SPLINE
SPL {X  -158.898, Y  +690.164, Z    +0.000, E1   +18.236, E3 -481675.354}
SPL {X  -159.149, Y  +687.882, Z    +0.000, E1   +16.368, E3 -481682.641}
SPL {X  -159.987, Y  +672.488, Z    +0.000, E1    +5.638, E3 -481704.183}
SPL {X  -159.990, Y  +663.928, Z    +0.000, E1    -0.338, E3 -481709.978}
SPL {X  -159.990, Y  +658.009, Z    +0.000, E1    -4.774, E3 -481713.678}
SPL {X  -159.990, Y  +651.567, Z    +0.000, E1    -9.674, E3 -481719.081}
SPL {X  -159.990, Y  +637.762, Z    +0.000, E1   -18.345, E3 -481736.439}
SPL {X  -159.990, Y  +626.382, Z    +0.000, E1   -22.040, E3 -481768.488}
SPL {X  -159.990, Y  +623.760, Z    +0.000, E1   -22.031, E3 -481782.266}
SPL {X  -159.990, Y  +621.334, Z    +0.000, E1   -22.029, E3 -481794.993}
SPL {X  -159.990, Y  +619.505, Z    +0.000, E1   -22.018, E3 -481804.608}
SPL {X  -159.990, Y  +617.621, Z    +0.000, E1   -22.025, E3 -481814.474}
SPL {X  -159.990, Y  +615.830, Z    +0.000, E1   -22.023, E3 -481823.874}
SPL {X  -159.990, Y  +614.007, Z    +0.000, E1   -22.018, E3 -481833.452}
SPL {X  -159.990, Y  +611.459, Z    +0.000, E1   -22.053, E3 -481846.738}
SPL {X  -159.990, Y  +608.810, Z    +0.000, E1   -22.023, E3 -481860.706}
SPL {X  -159.990, Y  +606.481, Z    +0.000, E1   -22.033, E3 -481872.882}
SPL {X  -159.990, Y  +603.419, Z    +0.000, E1   -22.064, E3 -481888.821}
SPL {X  -159.990, Y  +600.642, Z    +0.000, E1   -22.032, E3 -481903.451}
SPL {X  -159.990, Y  +598.568, Z    +0.000, E1   -22.046, E3 -481914.243}
SPL {X  -159.990, Y  +596.440, Z    +0.000, E1   -22.036, E3 -481925.425}
SPL {X  -159.990, Y  +593.768, Z    +0.000, E1   -22.071, E3 -481939.358}
SPL {X  -159.990, Y  +590.068, Z    +0.000, E1   -22.076, E3 -481958.726}
SPL {X  -159.990, Y  +587.130, Z    +0.000, E1   -22.046, E3 -481974.163}
SPL {X  -159.990, Y  +585.120, Z    +0.000, E1   -22.045, E3 -481984.665}
SPL {X  -159.990, Y  +583.118, Z    +0.000, E1   -22.052, E3 -481995.151}
SPL {X  -159.990, Y  +580.862, Z    +0.000, E1   -22.049, E3 -482006.989}
SPL {X  -159.990, Y  +578.386, Z    +0.000, E1   -22.057, E3 -482019.944}
SPL {X  -159.990, Y  +576.252, Z    +0.000, E1   -22.038, E3 -482031.168}
SPL {X  -159.990, Y  +574.280, Z    +0.000, E1   -22.051, E3 -482041.462}
SPL {X  -159.990, Y  +571.711, Z    +0.000, E1   -22.058, E3 -482054.935}
SPL {X  -159.990, Y  +569.285, Z    +0.000, E1   -22.044, E3 -482067.660}
SPL {X  -159.990, Y  +567.211, Z    +0.000, E1   -22.046, E3 -482078.522}
SPL {X  -159.990, Y  +565.039, Z    +0.000, E1   -22.047, E3 -482089.899}
SPL {X  -159.990, Y  +562.755, Z    +0.000, E1   -22.047, E3 -482101.884}
SPL {X  -159.990, Y  +559.661, Z    +0.000, E1   -22.078, E3 -482118.016}
SPL {X  -159.990, Y  +555.965, Z    +0.000, E1   -22.085, E3 -482137.325}
SPL {X  -159.990, Y  +553.115, Z    +0.000, E1   -22.054, E3 -482152.311}
SPL {X  -159.990, Y  +550.886, Z    +0.000, E1   -22.056, E3 -482163.992}
SPL {X  -159.990, Y  +547.986, Z    +0.000, E1   -22.078, E3 -482179.111}
SPL {X  -159.990, Y  +545.350, Z    +0.000, E1   -22.053, E3 -482192.973}
SPL {X  -159.990, Y  +543.405, Z    +0.000, E1   -22.048, E3 -482203.186}
SPL {X  -159.990, Y  +541.673, Z    +0.000, E1   -22.053, E3 -482212.249}
SPL {X  -159.990, Y  +539.341, Z    +0.000, E1   -22.056, E3 -482224.455}
SPL {X  -159.990, Y  +536.301, Z    +0.000, E1   -22.084, E3 -482240.309}
SPL {X  -159.990, Y  +533.389, Z    +0.000, E1   -22.057, E3 -482255.617}
SPL {X  -159.990, Y  +531.347, Z    +0.000, E1   -22.052, E3 -482266.317}
SPL {X  -159.990, Y  +529.626, Z    +0.000, E1   -22.051, E3 -482275.315}
SPL {X  -159.990, Y  +527.412, Z    +0.000, E1   -22.067, E3 -482286.867}
SPL {X  -159.990, Y  +524.425, Z    +0.000, E1   -22.078, E3 -482302.500}
SPL {X  -159.990, Y  +521.599, Z    +0.000, E1   -22.060, E3 -482317.342}
SPL {X  -159.990, Y  +519.209, Z    +0.000, E1   -22.063, E3 -482329.817}
SPL {X  -159.990, Y  +516.651, Z    +0.000, E1   -22.071, E3 -482343.196}
SPL {X  -159.990, Y  +514.122, Z    +0.000, E1   -22.061, E3 -482356.468}
SPL {X  -159.990, Y  +511.670, Z    +0.000, E1   -22.064, E3 -482369.318}
SPL {X  -159.990, Y  +506.947, Z    +0.000, E1   -23.726, E3 -482379.347}
SPL {X  -159.990, Y  +496.921, Z    +0.000, E1   -28.340, E3 -482388.095}
SPL {X  -159.990, Y  +495.822, Z    +0.000, E1   -27.449, E3 -482398.843}
SPL {X  -159.990, Y  +494.952, Z    +0.000, E1   -26.628, E3 -482408.426}
SPL {X  -159.990, Y  +493.896, Z    +0.000, E1   -25.736, E3 -482419.756}
SPL {X  -159.990, Y  +491.647, Z    +0.000, E1   -25.401, E3 -482432.291}
SPL {X  -159.990, Y  +488.807, Z    +0.000, E1   -25.397, E3 -482444.990}
SPL {X  -159.990, Y  +486.070, Z    +0.000, E1   -25.399, E3 -482457.221}
SPL {X  -159.990, Y  +483.747, Z    +0.000, E1   -25.384, E3 -482467.634}
SPL {X  -159.990, Y  +481.038, Z    +0.000, E1   -25.412, E3 -482479.689}
SPL {X  -159.990, Y  +478.407, Z    +0.000, E1   -25.384, E3 -482491.503}
SPL {X  -159.990, Y  +475.940, Z    +0.000, E1   -25.403, E3 -482502.493}
SPL {X  -159.990, Y  +473.026, Z    +0.000, E1   -25.399, E3 -482515.523}
SPL {X  -159.990, Y  +470.047, Z    +0.000, E1   -25.402, E3 -482528.842}
SPL {X  -159.990, Y  +467.082, Z    +0.000, E1   -25.399, E3 -482542.089}
SPL {X  -159.990, Y  +464.919, Z    +0.000, E1   -25.381, E3 -482551.815}
SPL {X  -159.990, Y  +462.520, Z    +0.000, E1   -25.400, E3 -482562.490}
SPL {X  -159.990, Y  +460.081, Z    +0.000, E1   -25.390, E3 -482573.391}
SPL {X  -159.990, Y  +457.497, Z    +0.000, E1   -25.403, E3 -482584.916}
SPL {X  -159.990, Y  +454.323, Z    +0.000, E1   -25.412, E3 -482599.075}
SPL {X  -159.990, Y  +450.823, Z    +0.000, E1   -25.417, E3 -482614.704}
SPL {X  -159.990, Y  +446.894, Z    +0.000, E1   -25.428, E3 -482632.261}
SPL {X  -159.990, Y  +443.345, Z    +0.000, E1   -25.390, E3 -482648.268}
SPL {X  -159.990, Y  +441.077, Z    +0.000, E1   -25.369, E3 -482658.466}
SPL {X  -159.990, Y  +438.608, Z    +0.000, E1   -25.392, E3 -482669.463}
SPL {X  -159.990, Y  +435.579, Z    +0.000, E1   -25.386, E3 -482683.017}
SPL {X  -159.990, Y  +432.613, Z    +0.000, E1   -25.390, E3 -482696.285}
SPL {X  -159.990, Y  +429.079, Z    +0.000, E1   -25.407, E3 -482712.055}
SPL {X  -159.990, Y  +426.149, Z    +0.000, E1   -25.374, E3 -482725.217}
SPL {X  -159.990, Y  +423.417, Z    +0.000, E1   -25.400, E3 -482737.383}
SPL {X  -159.990, Y  +420.283, Z    +0.000, E1   -25.386, E3 -482751.427}
SPL {X  -159.990, Y  +417.514, Z    +0.000, E1   -25.386, E3 -482763.812}
SPL {X  -159.990, Y  +414.805, Z    +0.000, E1   -25.385, E3 -482775.932}
SPL {X  -159.990, Y  +411.282, Z    +0.000, E1   -25.413, E3 -482791.632}
SPL {X  -159.990, Y  +407.450, Z    +0.000, E1   -25.401, E3 -482808.782}
SPL {X  -159.990, Y  +403.513, Z    +0.000, E1   -25.420, E3 -482826.335}
SPL {X  -159.990, Y  +399.257, Z    +0.000, E1   -25.420, E3 -482845.376}
SPL {X  -159.990, Y  +395.992, Z    +0.000, E1   -25.380, E3 -482860.066}
SPL {X  -159.990, Y  +393.569, Z    +0.000, E1   -25.379, E3 -482870.909}
SPL {X  -159.990, Y  +390.564, Z    +0.000, E1   -25.393, E3 -482884.353}
SPL {X  -159.990, Y  +387.503, Z    +0.000, E1   -25.378, E3 -482898.068}
SPL {X  -159.990, Y  +384.900, Z    +0.000, E1   -25.383, E3 -482909.678}
SPL {X  -159.990, Y  +382.110, Z    +0.000, E1   -25.393, E3 -482922.124}
SPL {X  -159.961, Y  +379.439, Z    +0.000, E1   -25.380, E3 -482934.103}
SPL {X  -159.894, Y  +376.959, Z    +0.000, E1   -25.370, E3 -482945.281}
SPL {X  -159.784, Y  +374.382, Z    +0.000, E1   -25.356, E3 -482956.921}
SPL {X  -159.621, Y  +371.640, Z    +0.000, E1   -25.335, E3 -482969.361}
SPL {X  -159.406, Y  +368.844, Z    +0.000, E1   -25.307, E3 -482982.074}
SPL {X  -159.144, Y  +366.072, Z    +0.000, E1   -25.281, E3 -482994.682}
SPL {X  -158.822, Y  +363.200, Z    +0.000, E1   -25.236, E3 -483007.855}
SPL {X  -158.491, Y  +360.654, Z    +0.000, E1   -25.188, E3 -483019.595}
SPL {X  -158.127, Y  +358.155, Z    +0.000, E1   -25.126, E3 -483031.214}
SPL {X  -158.095, Y  +357.947, Z    +0.000, E1   -21.741, E3 -483062.786}
ENDSPLINE

SPLINE
SPL {X  -158.454, Y  +360.384, Z    +0.000, E1   -19.366, E3 -483074.937}
SPL {X  -159.737, Y  +373.507, Z    +0.000, E1   -10.311, E3 -483096.973}
SPL {X  -159.990, Y  +382.574, Z    +0.000, E1    -4.463, E3 -483103.661}
SPL {X  -159.990, Y  +387.496, Z    +0.000, E1    -1.004, E3 -483106.406}
SPL {X  -159.990, Y  +395.121, Z    +0.000, E1    +4.514, E3 -483110.718}
SPL {X  -159.990, Y  +407.941, Z    +0.000, E1   +14.126, E3 -483122.792}
SPL {X  -159.990, Y  +418.671, Z    +0.000, E1   +19.855, E3 -483142.208}
SPL {X  -159.990, Y  +429.878, Z    +0.000, E1   +23.330, E3 -483172.264}
SPL {X  -159.990, Y  +432.103, Z    +0.000, E1   +23.301, E3 -483183.282}
SPL {X  -159.990, Y  +434.188, Z    +0.000, E1   +23.325, E3 -483193.479}
SPL {X  -159.990, Y  +436.320, Z    +0.000, E1   +23.304, E3 -483204.031}
SPL {X  -159.990, Y  +439.169, Z    +0.000, E1   +23.353, E3 -483217.948}
SPL {X  -159.990, Y  +442.945, Z    +0.000, E1   +23.339, E3 -483236.566}
SPL {X  -159.990, Y  +446.037, Z    +0.000, E1   +23.324, E3 -483251.816}
SPL {X  -159.990, Y  +448.797, Z    +0.000, E1   +23.331, E3 -483265.347}
SPL {X  -159.990, Y  +451.747, Z    +0.000, E1   +23.333, E3 -483279.895}
SPL {X  -159.990, Y  +455.185, Z    +0.000, E1   +23.350, E3 -483296.755}
SPL {X  -159.990, Y  +458.265, Z    +0.000, E1   +23.328, E3 -483311.941}
SPL {X  -159.990, Y  +460.492, Z    +0.000, E1   +23.317, E3 -483322.940}
SPL {X  -159.990, Y  +462.929, Z    +0.000, E1   +23.331, E3 -483334.896}
SPL {X  -159.990, Y  +465.027, Z    +0.000, E1   +23.313, E3 -483345.249}
SPL {X  -159.990, Y  +466.881, Z    +0.000, E1   +23.322, E3 -483354.359}
SPL {X  -159.990, Y  +468.951, Z    +0.000, E1   +23.319, E3 -483364.551}
SPL {X  -159.990, Y  +471.818, Z    +0.000, E1   +23.351, E3 -483378.597}
SPL {X  -159.990, Y  +474.801, Z    +0.000, E1   +23.320, E3 -483393.373}
SPL {X  -159.990, Y  +476.830, Z    +0.000, E1   +23.323, E3 -483403.352}
SPL {X  -159.990, Y  +479.553, Z    +0.000, E1   +23.328, E3 -483416.754}
SPL {X  -159.990, Y  +481.893, Z    +0.000, E1   +23.312, E3 -483428.304}
SPL {X  -159.990, Y  +483.782, Z    +0.000, E1   +23.316, E3 -483437.590}
SPL {X  -159.990, Y  +486.109, Z    +0.000, E1   +23.322, E3 -483449.042}
SPL {X  -159.990, Y  +489.247, Z    +0.000, E1   +23.348, E3 -483464.430}
SPL {X  -159.990, Y  +493.031, Z    +0.000, E1   +23.350, E3 -483483.054}
SPL {X  -159.990, Y  +496.869, Z    +0.000, E1   +23.349, E3 -483501.944}
SPL {X  -159.990, Y  +499.995, Z    +0.000, E1   +23.324, E3 -483517.377}
SPL {X  -159.990, Y  +502.456, Z    +0.000, E1   +23.324, E3 -483529.492}
SPL {X  -159.990, Y  +505.646, Z    +0.000, E1   +23.350, E3 -483545.147}
SPL {X  -159.990, Y  +508.862, Z    +0.000, E1   +23.328, E3 -483561.011}
SPL {X  -159.990, Y  +510.971, Z    +0.000, E1   +23.308, E3 -483571.439}
SPL {X  -159.990, Y  +512.484, Z    +0.000, E1   +23.309, E3 -483578.888}
SPL {X  -159.990, Y  +514.757, Z    +0.000, E1   +23.329, E3 -483590.041}
SPL {X  -159.990, Y  +517.536, Z    +0.000, E1   +23.326, E3 -483603.707}
SPL {X  -159.990, Y  +519.961, Z    +0.000, E1   +23.334, E3 -483615.560}
SPL {X  -159.990, Y  +521.849, Z    +0.000, E1   +23.320, E3 -483624.882}
SPL {X  -159.990, Y  +523.968, Z    +0.000, E1   +23.332, E3 -483635.318}
SPL {X  -159.990, Y  +526.466, Z    +0.000, E1   +23.320, E3 -483647.662}
SPL {X  -159.990, Y  +528.815, Z    +0.000, E1   +23.322, E3 -483659.221}
SPL {X  -159.990, Y  +531.246, Z    +0.000, E1   +23.325, E3 -483671.160}
SPL {X  -159.990, Y  +533.354, Z    +0.000, E1   +23.318, E3 -483681.545}
SPL {X  -159.990, Y  +534.931, Z    +0.000, E1   +23.312, E3 -483689.339}
SPL {X  -159.990, Y  +537.024, Z    +0.000, E1   +23.321, E3 -483699.638}
SPL {X  -159.990, Y  +539.129, Z    +0.000, E1   +23.310, E3 -483710.021}
SPL {X  -159.990, Y  +541.183, Z    +0.000, E1   +23.319, E3 -483720.118}
SPL {X  -159.990, Y  +544.314, Z    +0.000, E1   +23.352, E3 -483735.446}
SPL {X  -159.990, Y  +548.126, Z    +0.000, E1   +23.354, E3 -483754.201}
SPL {X  -159.990, Y  +551.344, Z    +0.000, E1   +23.327, E3 -483770.093}
SPL {X  -159.990, Y  +553.642, Z    +0.000, E1   +23.319, E3 -483781.412}
SPL {X  -159.990, Y  +556.481, Z    +0.000, E1   +23.354, E3 -483795.319}
SPL {X  -159.990, Y  +559.475, Z    +0.000, E1   +23.321, E3 -483810.125}
SPL {X  -159.990, Y  +561.830, Z    +0.000, E1   +23.325, E3 -483821.709}
SPL {X  -159.990, Y  +564.273, Z    +0.000, E1   +23.325, E3 -483833.733}
SPL {X  -159.990, Y  +566.342, Z    +0.000, E1   +23.314, E3 -483843.938}
SPL {X  -159.990, Y  +568.849, Z    +0.000, E1   +23.338, E3 -483856.233}
SPL {X  -159.990, Y  +572.204, Z    +0.000, E1   +23.344, E3 -483872.728}
SPL {X  -159.990, Y  +575.097, Z    +0.000, E1   +23.325, E3 -483887.005}
SPL {X  -159.990, Y  +577.540, Z    +0.000, E1   +23.325, E3 -483899.034}
SPL {X  -159.990, Y  +580.312, Z    +0.000, E1   +23.340, E3 -483912.615}
SPL {X  -159.990, Y  +583.018, Z    +0.000, E1   +23.331, E3 -483925.920}
SPL {X  -159.990, Y  +585.165, Z    +0.000, E1   +23.322, E3 -483936.536}
SPL {X  -159.990, Y  +587.388, Z    +0.000, E1   +23.328, E3 -483947.448}
SPL {X  -159.990, Y  +589.763, Z    +0.000, E1   +23.328, E3 -483959.135}
SPL {X  -159.990, Y  +592.397, Z    +0.000, E1   +23.344, E3 -483972.016}
SPL {X  -159.990, Y  +594.928, Z    +0.000, E1   +23.334, E3 -483984.478}
SPL {X  -159.990, Y  +597.981, Z    +0.000, E1   +23.373, E3 -483999.393}
SPL {X  -159.990, Y  +600.935, Z    +0.000, E1   +23.343, E3 -484013.926}
SPL {X  -159.990, Y  +603.047, Z    +0.000, E1   +23.344, E3 -484024.311}
SPL {X  -159.990, Y  +605.187, Z    +0.000, E1   +23.344, E3 -484034.833}
SPL {X  -159.990, Y  +607.319, Z    +0.000, E1   +23.353, E3 -484045.295}
SPL {X  -159.990, Y  +610.569, Z    +0.000, E1   +23.372, E3 -484061.260}
SPL {X  -159.990, Y  +613.591, Z    +0.000, E1   +23.342, E3 -484076.189}
SPL {X  -159.990, Y  +615.604, Z    +0.000, E1   +23.330, E3 -484086.127}
SPL {X  -159.990, Y  +618.445, Z    +0.000, E1   +23.368, E3 -484100.040}
SPL {X  -159.990, Y  +621.517, Z    +0.000, E1   +23.337, E3 -484115.204}
SPL {X  -159.990, Y  +623.764, Z    +0.000, E1   +23.335, E3 -484126.255}
SPL {X  -159.990, Y  +625.941, Z    +0.000, E1   +23.337, E3 -484136.946}
SPL {X  -159.990, Y  +628.611, Z    +0.000, E1   +23.357, E3 -484150.025}
SPL {X  -159.990, Y  +631.169, Z    +0.000, E1   +23.338, E3 -484162.629}
SPL {X  -159.990, Y  +633.318, Z    +0.000, E1   +23.339, E3 -484173.218}
SPL {X  -159.990, Y  +635.650, Z    +0.000, E1   +23.339, E3 -484184.689}
SPL {X  -159.990, Y  +637.839, Z    +0.000, E1   +23.335, E3 -484195.500}
SPL {X  -159.990, Y  +640.072, Z    +0.000, E1   +23.325, E3 -484206.532}
SPL {X  -159.990, Y  +642.230, Z    +0.000, E1   +23.323, E3 -484217.213}
SPL {X  -159.990, Y  +645.287, Z    +0.000, E1   +23.340, E3 -484232.239}
SPL {X  -159.990, Y  +648.792, Z    +0.000, E1   +23.346, E3 -484249.498}
SPL {X  -159.990, Y  +652.623, Z    +0.000, E1   +23.348, E3 -484268.333}
SPL {X  -159.990, Y  +656.380, Z    +0.000, E1   +23.347, E3 -484286.827}
SPL {X  -159.990, Y  +659.180, Z    +0.000, E1   +23.314, E3 -484300.676}
SPL {X  -159.990, Y  +661.392, Z    +0.000, E1   +23.318, E3 -484311.569}
SPL {X  -159.990, Y  +663.662, Z    +0.000, E1   +23.322, E3 -484322.693}
SPL {X  -159.990, Y  +665.964, Z    +0.000, E1   +23.328, E3 -484333.984}
SPL {X  -159.990, Y  +668.989, Z    +0.000, E1   +23.359, E3 -484348.820}
SPL {X  -159.983, Y  +672.946, Z    +0.000, E1   +23.359, E3 -484368.301}
SPL {X  -159.924, Y  +676.110, Z    +0.000, E1   +23.320, E3 -484384.000}
SPL {X  -159.845, Y  +678.302, Z    +0.000, E1   +23.298, E3 -484394.902}
SPL {X  -159.760, Y  +680.081, Z    +0.000, E1   +23.288, E3 -484403.746}
SPL {X  -159.626, Y  +682.287, Z    +0.000, E1   +23.280, E3 -484414.717}
SPL {X  -159.462, Y  +684.486, Z    +0.000, E1   +23.258, E3 -484425.717}
SPL {X  -159.246, Y  +686.911, Z    +0.000, E1   +23.230, E3 -484437.878}
SPL {X  -159.019, Y  +689.098, Z    +0.000, E1   +23.200, E3 -484448.880}
SPL {X  -158.771, Y  +691.210, Z    +0.000, E1   +23.159, E3 -484459.555}
SPL {X  -158.553, Y  +692.896, Z    +0.000, E1   +23.130, E3 -484468.085}
ENDSPLINE

SPLINE
SPL {X  -158.898, Y  +690.164, Z    +0.000, E1   +18.236, E3 -484501.441}
SPL {X  -159.149, Y  +687.882, Z    +0.000, E1   +16.368, E3 -484508.728}
SPL {X  -159.987, Y  +672.488, Z    +0.000, E1    +5.638, E3 -484530.270}
SPL {X  -159.990, Y  +663.928, Z    +0.000, E1    -0.338, E3 -484536.065}
SPL {X  -159.990, Y  +658.009, Z    +0.000, E1    -4.774, E3 -484539.765}
SPL {X  -159.990, Y  +651.567, Z    +0.000, E1    -9.674, E3 -484545.168}
SPL {X  -159.990, Y  +638.711, Z    +0.000, E1   -17.883, E3 -484560.814}
SPL {X  -159.990, Y  +631.642, Z    +0.000, E1   -20.884, E3 -484576.373}
SPL {X  -159.990, Y  +626.048, Z    +0.000, E1   -22.026, E3 -484596.366}
SPL {X  -159.990, Y  +623.760, Z    +0.000, E1   -22.031, E3 -484608.353}
SPL {X  -159.990, Y  +621.334, Z    +0.000, E1   -22.029, E3 -484621.080}
SPL {X  -159.990, Y  +619.505, Z    +0.000, E1   -22.018, E3 -484630.695}
SPL {X  -159.990, Y  +617.621, Z    +0.000, E1   -22.025, E3 -484640.561}
SPL {X  -159.990, Y  +615.830, Z    +0.000, E1   -22.023, E3 -484649.961}
SPL {X  -159.990, Y  +613.034, Z    +0.000, E1   -22.053, E3 -484664.568}
SPL {X  -159.990, Y  +609.503, Z    +0.000, E1   -22.054, E3 -484683.094}
SPL {X  -159.990, Y  +605.804, Z    +0.000, E1   -22.064, E3 -484702.438}
SPL {X  -159.990, Y  +602.819, Z    +0.000, E1   -22.037, E3 -484718.110}
SPL {X  -159.990, Y  +600.642, Z    +0.000, E1   -22.032, E3 -484729.538}
SPL {X  -159.990, Y  +598.568, Z    +0.000, E1   -22.046, E3 -484740.330}
SPL {X  -159.990, Y  +595.493, Z    +0.000, E1   -22.070, E3 -484756.414}
SPL {X  -159.990, Y  +592.865, Z    +0.000, E1   -22.036, E3 -484770.242}
SPL {X  -159.990, Y  +590.803, Z    +0.000, E1   -22.046, E3 -484781.033}
SPL {X  -159.990, Y  +587.778, Z    +0.000, E1   -22.073, E3 -484796.808}
SPL {X  -159.990, Y  +585.120, Z    +0.000, E1   -22.045, E3 -484810.752}
SPL {X  -159.990, Y  +583.118, Z    +0.000, E1   -22.052, E3 -484821.238}
SPL {X  -159.990, Y  +580.131, Z    +0.000, E1   -22.078, E3 -484836.845}
SPL {X  -159.990, Y  +576.888, Z    +0.000, E1   -22.061, E3 -484853.875}
SPL {X  -159.990, Y  +574.280, Z    +0.000, E1   -22.051, E3 -484867.549}
SPL {X  -159.990, Y  +572.375, Z    +0.000, E1   -22.037, E3 -484877.587}
SPL {X  -159.990, Y  +569.881, Z    +0.000, E1   -22.067, E3 -484890.581}
SPL {X  -159.990, Y  +567.211, Z    +0.000, E1   -22.046, E3 -484904.609}
SPL {X  -159.990, Y  +565.039, Z    +0.000, E1   -22.047, E3 -484915.986}
SPL {X  -159.990, Y  +562.755, Z    +0.000, E1   -22.047, E3 -484927.971}
SPL {X  -159.990, Y  +559.661, Z    +0.000, E1   -22.078, E3 -484944.103}
SPL {X  -159.990, Y  +555.965, Z    +0.000, E1   -22.085, E3 -484963.412}
SPL {X  -159.990, Y  +553.115, Z    +0.000, E1   -22.054, E3 -484978.398}
SPL {X  -159.990, Y  +550.886, Z    +0.000, E1   -22.056, E3 -484990.079}
SPL {X  -159.990, Y  +547.986, Z    +0.000, E1   -22.078, E3 -485005.198}
SPL {X  -159.990, Y  +545.350, Z    +0.000, E1   -22.053, E3 -485019.060}
SPL {X  -159.990, Y  +543.405, Z    +0.000, E1   -22.048, E3 -485029.273}
SPL {X  -159.990, Y  +541.673, Z    +0.000, E1   -22.053, E3 -485038.336}
SPL {X  -159.990, Y  +539.341, Z    +0.000, E1   -22.056, E3 -485050.542}
SPL {X  -159.990, Y  +536.301, Z    +0.000, E1   -22.084, E3 -485066.396}
SPL {X  -159.990, Y  +533.389, Z    +0.000, E1   -22.057, E3 -485081.704}
SPL {X  -159.990, Y  +530.476, Z    +0.000, E1   -22.084, E3 -485096.891}
SPL {X  -159.990, Y  +527.412, Z    +0.000, E1   -22.067, E3 -485112.954}
SPL {X  -159.990, Y  +525.349, Z    +0.000, E1   -22.050, E3 -485123.795}
SPL {X  -159.990, Y  +523.717, Z    +0.000, E1   -22.050, E3 -485132.361}
SPL {X  -159.990, Y  +521.599, Z    +0.000, E1   -22.060, E3 -485143.429}
SPL {X  -159.990, Y  +519.209, Z    +0.000, E1   -22.063, E3 -485155.904}
SPL {X  -159.990, Y  +517.330, Z    +0.000, E1   -22.053, E3 -485165.760}
SPL {X  -159.990, Y  +514.729, Z    +0.000, E1   -22.089, E3 -485179.318}
SPL {X  -159.990, Y  +511.670, Z    +0.000, E1   -22.064, E3 -485195.405}
SPL {X  -159.990, Y  +506.947, Z    +0.000, E1   -23.726, E3 -485205.434}
SPL {X  -159.990, Y  +496.921, Z    +0.000, E1   -28.340, E3 -485214.182}
SPL {X  -159.990, Y  +495.822, Z    +0.000, E1   -27.449, E3 -485224.930}
SPL {X  -159.990, Y  +494.952, Z    +0.000, E1   -26.628, E3 -485234.513}
SPL {X  -159.990, Y  +493.896, Z    +0.000, E1   -25.736, E3 -485245.843}
SPL {X  -159.990, Y  +491.647, Z    +0.000, E1   -25.401, E3 -485258.378}
SPL {X  -159.990, Y  +488.807, Z    +0.000, E1   -25.397, E3 -485271.077}
SPL {X  -159.990, Y  +486.070, Z    +0.000, E1   -25.399, E3 -485283.308}
SPL {X  -159.990, Y  +482.821, Z    +0.000, E1   -25.411, E3 -485297.809}
SPL {X  -159.990, Y  +480.183, Z    +0.000, E1   -25.384, E3 -485309.650}
SPL {X  -159.990, Y  +477.508, Z    +0.000, E1   -25.410, E3 -485321.558}
SPL {X  -159.990, Y  +473.634, Z    +0.000, E1   -25.426, E3 -485338.848}
SPL {X  -159.990, Y  +470.047, Z    +0.000, E1   -25.402, E3 -485354.928}
SPL {X  -159.990, Y  +466.213, Z    +0.000, E1   -25.433, E3 -485372.008}
SPL {X  -159.990, Y  +462.520, Z    +0.000, E1   -25.400, E3 -485388.577}
SPL {X  -159.990, Y  +460.081, Z    +0.000, E1   -25.390, E3 -485399.478}
SPL {X  -159.990, Y  +457.497, Z    +0.000, E1   -25.403, E3 -485411.003}
SPL {X  -159.990, Y  +455.126, Z    +0.000, E1   -25.389, E3 -485421.611}
SPL {X  -159.990, Y  +452.123, Z    +0.000, E1   -25.426, E3 -485434.969}
SPL {X  -159.990, Y  +448.503, Z    +0.000, E1   -25.410, E3 -485451.170}
SPL {X  -159.990, Y  +445.882, Z    +0.000, E1   -25.385, E3 -485462.973}
SPL {X  -159.990, Y  +443.345, Z    +0.000, E1   -25.390, E3 -485474.355}
SPL {X  -159.990, Y  +441.077, Z    +0.000, E1   -25.369, E3 -485484.553}
SPL {X  -159.990, Y  +438.608, Z    +0.000, E1   -25.392, E3 -485495.550}
SPL {X  -159.990, Y  +434.852, Z    +0.000, E1   -25.415, E3 -485512.305}
SPL {X  -159.990, Y  +430.645, Z    +0.000, E1   -25.414, E3 -485531.124}
SPL {X  -159.990, Y  +426.865, Z    +0.000, E1   -25.398, E3 -485548.054}
SPL {X  -159.990, Y  +424.251, Z    +0.000, E1   -25.375, E3 -485559.791}
SPL {X  -159.990, Y  +421.010, Z    +0.000, E1   -25.418, E3 -485574.206}
SPL {X  -159.990, Y  +417.514, Z    +0.000, E1   -25.386, E3 -485589.899}
SPL {X  -159.990, Y  +414.805, Z    +0.000, E1   -25.385, E3 -485602.019}
SPL {X  -159.990, Y  +411.282, Z    +0.000, E1   -25.413, E3 -485617.719}
SPL {X  -159.990, Y  +408.351, Z    +0.000, E1   -25.372, E3 -485630.906}
SPL {X  -159.990, Y  +405.773, Z    +0.000, E1   -25.398, E3 -485642.359}
SPL {X  -159.990, Y  +402.805, Z    +0.000, E1   -25.389, E3 -485655.645}
SPL {X  -159.990, Y  +400.083, Z    +0.000, E1   -25.388, E3 -485667.822}
SPL {X  -159.990, Y  +396.740, Z    +0.000, E1   -25.410, E3 -485682.746}
SPL {X  -159.990, Y  +392.622, Z    +0.000, E1   -25.413, E3 -485701.174}
SPL {X  -159.990, Y  +388.328, Z    +0.000, E1   -25.413, E3 -485720.402}
SPL {X  -159.990, Y  +384.900, Z    +0.000, E1   -25.383, E3 -485735.764}
SPL {X  -159.990, Y  +382.110, Z    +0.000, E1   -25.393, E3 -485748.211}
SPL {X  -159.961, Y  +379.439, Z    +0.000, E1   -25.380, E3 -485760.190}
SPL {X  -159.894, Y  +376.959, Z    +0.000, E1   -25.370, E3 -485771.368}
SPL {X  -159.784, Y  +374.382, Z    +0.000, E1   -25.356, E3 -485783.008}
SPL {X  -159.621, Y  +371.640, Z    +0.000, E1   -25.335, E3 -485795.448}
SPL {X  -159.406, Y  +368.844, Z    +0.000, E1   -25.307, E3 -485808.161}
SPL {X  -159.144, Y  +366.072, Z    +0.000, E1   -25.281, E3 -485820.769}
SPL {X  -158.822, Y  +363.200, Z    +0.000, E1   -25.236, E3 -485833.941}
SPL {X  -158.491, Y  +360.654, Z    +0.000, E1   -25.188, E3 -485845.682}
SPL {X  -158.127, Y  +358.155, Z    +0.000, E1   -25.126, E3 -485857.301}
SPL {X  -158.095, Y  +357.947, Z    +0.000, E1   -21.741, E3 -485888.873}
ENDSPLINE

SPLINE
SPL {X  -158.454, Y  +360.384, Z    +0.000, E1   -19.366, E3 -485901.024}
SPL {X  -159.737, Y  +373.507, Z    +0.000, E1   -10.311, E3 -485923.060}
SPL {X  -159.990, Y  +382.574, Z    +0.000, E1    -4.463, E3 -485929.748}
SPL {X  -159.990, Y  +389.909, Z    +0.000, E1    +0.662, E3 -485933.762}
SPL {X  -159.990, Y  +396.289, Z    +0.000, E1    +5.500, E3 -485937.542}
SPL {X  -159.990, Y  +407.941, Z    +0.000, E1   +14.126, E3 -485948.879}
SPL {X  -159.990, Y  +418.671, Z    +0.000, E1   +19.855, E3 -485968.295}
SPL {X  -159.990, Y  +429.878, Z    +0.000, E1   +23.330, E3 -485998.350}
SPL {X  -159.990, Y  +432.103, Z    +0.000, E1   +23.301, E3 -486009.369}
SPL {X  -159.990, Y  +434.188, Z    +0.000, E1   +23.325, E3 -486019.566}
SPL {X  -159.990, Y  +437.007, Z    +0.000, E1   +23.323, E3 -486033.457}
SPL {X  -159.990, Y  +439.778, Z    +0.000, E1   +23.323, E3 -486047.089}
SPL {X  -159.990, Y  +442.010, Z    +0.000, E1   +23.308, E3 -486058.110}
SPL {X  -159.990, Y  +443.729, Z    +0.000, E1   +23.310, E3 -486066.566}
SPL {X  -159.990, Y  +446.037, Z    +0.000, E1   +23.324, E3 -486077.903}
SPL {X  -159.990, Y  +449.434, Z    +0.000, E1   +23.356, E3 -486094.525}
SPL {X  -159.990, Y  +453.256, Z    +0.000, E1   +23.349, E3 -486113.360}
SPL {X  -159.990, Y  +455.953, Z    +0.000, E1   +23.320, E3 -486126.674}
SPL {X  -159.990, Y  +458.265, Z    +0.000, E1   +23.328, E3 -486138.028}
SPL {X  -159.990, Y  +461.258, Z    +0.000, E1   +23.344, E3 -486152.744}
SPL {X  -159.990, Y  +464.382, Z    +0.000, E1   +23.332, E3 -486168.126}
SPL {X  -159.990, Y  +466.881, Z    +0.000, E1   +23.322, E3 -486180.446}
SPL {X  -159.990, Y  +468.951, Z    +0.000, E1   +23.319, E3 -486190.638}
SPL {X  -159.990, Y  +470.991, Z    +0.000, E1   +23.322, E3 -486200.668}
SPL {X  -159.990, Y  +474.027, Z    +0.000, E1   +23.352, E3 -486215.571}
SPL {X  -159.990, Y  +477.600, Z    +0.000, E1   +23.351, E3 -486233.175}
SPL {X  -159.990, Y  +481.169, Z    +0.000, E1   +23.337, E3 -486250.772}
SPL {X  -159.990, Y  +483.782, Z    +0.000, E1   +23.316, E3 -486263.677}
SPL {X  -159.990, Y  +486.109, Z    +0.000, E1   +23.322, E3 -486275.129}
SPL {X  -159.990, Y  +489.247, Z    +0.000, E1   +23.348, E3 -486290.517}
SPL {X  -159.990, Y  +493.031, Z    +0.000, E1   +23.350, E3 -486309.141}
SPL {X  -159.990, Y  +496.869, Z    +0.000, E1   +23.349, E3 -486328.031}
SPL {X  -159.990, Y  +499.995, Z    +0.000, E1   +23.324, E3 -486343.464}
SPL {X  -159.990, Y  +502.456, Z    +0.000, E1   +23.324, E3 -486355.579}
SPL {X  -159.990, Y  +505.646, Z    +0.000, E1   +23.350, E3 -486371.234}
SPL {X  -159.990, Y  +508.862, Z    +0.000, E1   +23.328, E3 -486387.098}
SPL {X  -159.990, Y  +510.971, Z    +0.000, E1   +23.308, E3 -486397.526}
SPL {X  -159.990, Y  +513.289, Z    +0.000, E1   +23.332, E3 -486408.893}
SPL {X  -159.990, Y  +516.860, Z    +0.000, E1   +23.355, E3 -486426.410}
SPL {X  -159.990, Y  +520.719, Z    +0.000, E1   +23.363, E3 -486445.320}
SPL {X  -159.990, Y  +523.968, Z    +0.000, E1   +23.332, E3 -486461.405}
SPL {X  -159.990, Y  +526.466, Z    +0.000, E1   +23.320, E3 -486473.748}
SPL {X  -159.990, Y  +528.815, Z    +0.000, E1   +23.322, E3 -486485.308}
SPL {X  -159.990, Y  +531.246, Z    +0.000, E1   +23.325, E3 -486497.247}
SPL {X  -159.990, Y  +534.143, Z    +0.000, E1   +23.341, E3 -486511.482}
SPL {X  -159.990, Y  +537.024, Z    +0.000, E1   +23.321, E3 -486525.725}
SPL {X  -159.990, Y  +539.129, Z    +0.000, E1   +23.310, E3 -486536.108}
SPL {X  -159.990, Y  +541.882, Z    +0.000, E1   +23.346, E3 -486549.589}
SPL {X  -159.990, Y  +544.941, Z    +0.000, E1   +23.325, E3 -486564.671}
SPL {X  -159.990, Y  +547.390, Z    +0.000, E1   +23.325, E3 -486576.725}
SPL {X  -159.990, Y  +550.708, Z    +0.000, E1   +23.357, E3 -486592.992}
SPL {X  -159.990, Y  +553.642, Z    +0.000, E1   +23.319, E3 -486607.499}
SPL {X  -159.990, Y  +555.637, Z    +0.000, E1   +23.323, E3 -486617.313}
SPL {X  -159.990, Y  +558.758, Z    +0.000, E1   +23.351, E3 -486632.623}
SPL {X  -159.990, Y  +561.830, Z    +0.000, E1   +23.325, E3 -486647.796}
SPL {X  -159.990, Y  +564.273, Z    +0.000, E1   +23.325, E3 -486659.820}
SPL {X  -159.990, Y  +567.351, Z    +0.000, E1   +23.348, E3 -486674.916}
SPL {X  -159.990, Y  +570.560, Z    +0.000, E1   +23.333, E3 -486690.746}
SPL {X  -159.990, Y  +572.975, Z    +0.000, E1   +23.316, E3 -486702.665}
SPL {X  -159.990, Y  +575.097, Z    +0.000, E1   +23.325, E3 -486713.092}
SPL {X  -159.990, Y  +578.356, Z    +0.000, E1   +23.358, E3 -486729.064}
SPL {X  -159.990, Y  +582.292, Z    +0.000, E1   +23.360, E3 -486748.380}
SPL {X  -159.990, Y  +585.165, Z    +0.000, E1   +23.322, E3 -486762.623}
SPL {X  -159.990, Y  +587.388, Z    +0.000, E1   +23.328, E3 -486773.535}
SPL {X  -159.990, Y  +590.594, Z    +0.000, E1   +23.363, E3 -486789.227}
SPL {X  -159.990, Y  +594.301, Z    +0.000, E1   +23.358, E3 -486807.432}
SPL {X  -159.990, Y  +597.981, Z    +0.000, E1   +23.373, E3 -486825.480}
SPL {X  -159.990, Y  +600.935, Z    +0.000, E1   +23.343, E3 -486840.012}
SPL {X  -159.990, Y  +603.047, Z    +0.000, E1   +23.344, E3 -486850.398}
SPL {X  -159.990, Y  +605.187, Z    +0.000, E1   +23.344, E3 -486860.920}
SPL {X  -159.990, Y  +607.319, Z    +0.000, E1   +23.353, E3 -486871.382}
SPL {X  -159.990, Y  +610.569, Z    +0.000, E1   +23.372, E3 -486887.347}
SPL {X  -159.990, Y  +613.591, Z    +0.000, E1   +23.342, E3 -486902.276}
SPL {X  -159.990, Y  +615.604, Z    +0.000, E1   +23.330, E3 -486912.214}
SPL {X  -159.990, Y  +618.445, Z    +0.000, E1   +23.368, E3 -486926.127}
SPL {X  -159.990, Y  +621.517, Z    +0.000, E1   +23.337, E3 -486941.291}
SPL {X  -159.990, Y  +623.764, Z    +0.000, E1   +23.335, E3 -486952.342}
SPL {X  -159.990, Y  +626.608, Z    +0.000, E1   +23.361, E3 -486966.267}
SPL {X  -159.990, Y  +630.271, Z    +0.000, E1   +23.375, E3 -486984.228}
SPL {X  -159.990, Y  +633.318, Z    +0.000, E1   +23.339, E3 -486999.305}
SPL {X  -159.990, Y  +635.650, Z    +0.000, E1   +23.339, E3 -487010.776}
SPL {X  -159.990, Y  +637.839, Z    +0.000, E1   +23.335, E3 -487021.587}
SPL {X  -159.990, Y  +640.072, Z    +0.000, E1   +23.325, E3 -487032.619}
SPL {X  -159.990, Y  +642.230, Z    +0.000, E1   +23.323, E3 -487043.300}
SPL {X  -159.990, Y  +645.287, Z    +0.000, E1   +23.340, E3 -487058.326}
SPL {X  -159.990, Y  +648.792, Z    +0.000, E1   +23.346, E3 -487075.585}
SPL {X  -159.990, Y  +652.623, Z    +0.000, E1   +23.348, E3 -487094.420}
SPL {X  -159.990, Y  +656.380, Z    +0.000, E1   +23.347, E3 -487112.914}
SPL {X  -159.990, Y  +659.180, Z    +0.000, E1   +23.314, E3 -487126.763}
SPL {X  -159.990, Y  +661.392, Z    +0.000, E1   +23.318, E3 -487137.656}
SPL {X  -159.990, Y  +663.662, Z    +0.000, E1   +23.322, E3 -487148.780}
SPL {X  -159.990, Y  +665.964, Z    +0.000, E1   +23.328, E3 -487160.071}
SPL {X  -159.990, Y  +668.989, Z    +0.000, E1   +23.359, E3 -487174.907}
SPL {X  -159.983, Y  +672.946, Z    +0.000, E1   +23.359, E3 -487194.388}
SPL {X  -159.924, Y  +676.110, Z    +0.000, E1   +23.320, E3 -487210.087}
SPL {X  -159.845, Y  +678.302, Z    +0.000, E1   +23.298, E3 -487220.989}
SPL {X  -159.760, Y  +680.081, Z    +0.000, E1   +23.288, E3 -487229.833}
SPL {X  -159.626, Y  +682.287, Z    +0.000, E1   +23.280, E3 -487240.804}
SPL {X  -159.462, Y  +684.486, Z    +0.000, E1   +23.258, E3 -487251.804}
SPL {X  -159.246, Y  +686.911, Z    +0.000, E1   +23.230, E3 -487263.965}
SPL {X  -159.019, Y  +689.098, Z    +0.000, E1   +23.200, E3 -487274.967}
SPL {X  -158.660, Y  +692.086, Z    +0.000, E1   +23.176, E3 -487290.011}
ENDSPLINE

SPLINE
SPL {X  -159.063, Y  +688.696, Z    +0.000, E1   +17.094, E3 -487332.293}
SPL {X  -159.987, Y  +672.488, Z    +0.000, E1    +5.638, E3 -487356.357}
SPL {X  -159.990, Y  +663.928, Z    +0.000, E1    -0.338, E3 -487362.152}
SPL {X  -159.990, Y  +658.009, Z    +0.000, E1    -4.774, E3 -487365.852}
SPL {X  -159.990, Y  +651.567, Z    +0.000, E1    -9.674, E3 -487371.255}
SPL {X  -159.990, Y  +638.711, Z    +0.000, E1   -17.883, E3 -487386.901}
SPL {X  -159.990, Y  +631.642, Z    +0.000, E1   -20.884, E3 -487402.460}
SPL {X  -159.990, Y  +626.048, Z    +0.000, E1   -22.026, E3 -487422.453}
SPL {X  -159.990, Y  +623.760, Z    +0.000, E1   -22.031, E3 -487434.440}
SPL {X  -159.990, Y  +621.334, Z    +0.000, E1   -22.029, E3 -487447.167}
SPL {X  -159.990, Y  +619.505, Z    +0.000, E1   -22.018, E3 -487456.782}
SPL {X  -159.990, Y  +617.621, Z    +0.000, E1   -22.025, E3 -487466.648}
SPL {X  -159.990, Y  +615.830, Z    +0.000, E1   -22.023, E3 -487476.048}
SPL {X  -159.990, Y  +613.034, Z    +0.000, E1   -22.053, E3 -487490.655}
SPL {X  -159.990, Y  +609.503, Z    +0.000, E1   -22.054, E3 -487509.181}
SPL {X  -159.990, Y  +605.804, Z    +0.000, E1   -22.064, E3 -487528.525}
SPL {X  -159.990, Y  +602.819, Z    +0.000, E1   -22.037, E3 -487544.197}
SPL {X  -159.990, Y  +600.642, Z    +0.000, E1   -22.032, E3 -487555.625}
SPL {X  -159.990, Y  +598.568, Z    +0.000, E1   -22.046, E3 -487566.417}
SPL {X  -159.990, Y  +595.493, Z    +0.000, E1   -22.070, E3 -487582.501}
SPL {X  -159.990, Y  +592.865, Z    +0.000, E1   -22.036, E3 -487596.329}
SPL {X  -159.990, Y  +590.803, Z    +0.000, E1   -22.046, E3 -487607.120}
SPL {X  -159.990, Y  +587.778, Z    +0.000, E1   -22.073, E3 -487622.895}
SPL {X  -159.990, Y  +585.120, Z    +0.000, E1   -22.045, E3 -487636.839}
SPL {X  -159.990, Y  +583.118, Z    +0.000, E1   -22.052, E3 -487647.325}
SPL {X  -159.990, Y  +580.862, Z    +0.000, E1   -22.049, E3 -487659.163}
SPL {X  -159.990, Y  +578.386, Z    +0.000, E1   -22.057, E3 -487672.118}
SPL {X  -159.990, Y  +576.252, Z    +0.000, E1   -22.038, E3 -487683.341}
SPL {X  -159.990, Y  +574.280, Z    +0.000, E1   -22.051, E3 -487693.635}
SPL {X  -159.990, Y  +571.711, Z    +0.000, E1   -22.058, E3 -487707.109}
SPL {X  -159.990, Y  +569.285, Z    +0.000, E1   -22.044, E3 -487719.834}
SPL {X  -159.990, Y  +567.211, Z    +0.000, E1   -22.046, E3 -487730.696}
SPL {X  -159.990, Y  +565.039, Z    +0.000, E1   -22.047, E3 -487742.073}
SPL {X  -159.990, Y  +562.755, Z    +0.000, E1   -22.047, E3 -487754.058}
SPL {X  -159.990, Y  +560.652, Z    +0.000, E1   -22.038, E3 -487765.103}
SPL {X  -159.990, Y  +558.852, Z    +0.000, E1   -22.046, E3 -487774.475}
SPL {X  -159.990, Y  +556.672, Z    +0.000, E1   -22.055, E3 -487785.865}
SPL {X  -159.990, Y  +553.726, Z    +0.000, E1   -22.080, E3 -487801.227}
SPL {X  -159.990, Y  +550.886, Z    +0.000, E1   -22.056, E3 -487816.166}
SPL {X  -159.990, Y  +548.814, Z    +0.000, E1   -22.049, E3 -487827.012}
SPL {X  -159.990, Y  +546.122, Z    +0.000, E1   -22.088, E3 -487841.025}
SPL {X  -159.990, Y  +542.390, Z    +0.000, E1   -22.086, E3 -487860.607}
SPL {X  -159.990, Y  +539.341, Z    +0.000, E1   -22.056, E3 -487876.629}
SPL {X  -159.990, Y  +536.301, Z    +0.000, E1   -22.084, E3 -487892.483}
SPL {X  -159.990, Y  +533.389, Z    +0.000, E1   -22.057, E3 -487907.791}
SPL {X  -159.990, Y  +531.347, Z    +0.000, E1   -22.052, E3 -487918.491}
SPL {X  -159.990, Y  +529.626, Z    +0.000, E1   -22.051, E3 -487927.488}
SPL {X  -159.990, Y  +527.412, Z    +0.000, E1   -22.067, E3 -487939.041}
SPL {X  -159.990, Y  +524.425, Z    +0.000, E1   -22.078, E3 -487954.674}
SPL {X  -159.990, Y  +521.599, Z    +0.000, E1   -22.060, E3 -487969.516}
SPL {X  -159.990, Y  +519.209, Z    +0.000, E1   -22.063, E3 -487981.991}
SPL {X  -159.990, Y  +516.651, Z    +0.000, E1   -22.071, E3 -487995.370}
SPL {X  -159.990, Y  +514.122, Z    +0.000, E1   -22.061, E3 -488008.642}
SPL {X  -159.990, Y  +511.670, Z    +0.000, E1   -22.064, E3 -488021.492}
SPL {X  -159.990, Y  +506.947, Z    +0.000, E1   -23.726, E3 -488031.520}
SPL {X  -159.990, Y  +496.921, Z    +0.000, E1   -28.340, E3 -488040.269}
SPL {X  -159.990, Y  +495.822, Z    +0.000, E1   -27.449, E3 -488051.017}
SPL {X  -159.990, Y  +494.952, Z    +0.000, E1   -26.628, E3 -488060.600}
SPL {X  -159.990, Y  +493.896, Z    +0.000, E1   -25.736, E3 -488071.930}
SPL {X  -159.990, Y  +491.647, Z    +0.000, E1   -25.401, E3 -488084.465}
SPL {X  -159.990, Y  +488.807, Z    +0.000, E1   -25.397, E3 -488097.164}
SPL {X  -159.990, Y  +486.070, Z    +0.000, E1   -25.399, E3 -488109.395}
SPL {X  -159.990, Y  +483.747, Z    +0.000, E1   -25.384, E3 -488119.808}
SPL {X  -159.990, Y  +481.038, Z    +0.000, E1   -25.412, E3 -488131.863}
SPL {X  -159.990, Y  +478.407, Z    +0.000, E1   -25.384, E3 -488143.677}
SPL {X  -159.990, Y  +475.940, Z    +0.000, E1   -25.403, E3 -488154.667}
SPL {X  -159.990, Y  +473.026, Z    +0.000, E1   -25.399, E3 -488167.697}
SPL {X  -159.990, Y  +470.047, Z    +0.000, E1   -25.402, E3 -488181.015}
SPL {X  -159.990, Y  +466.213, Z    +0.000, E1   -25.433, E3 -488198.095}
SPL {X  -159.990, Y  +462.520, Z    +0.000, E1   -25.400, E3 -488214.664}
SPL {X  -159.990, Y  +460.081, Z    +0.000, E1   -25.390, E3 -488225.565}
SPL {X  -159.990, Y  +457.497, Z    +0.000, E1   -25.403, E3 -488237.090}
SPL {X  -159.990, Y  +454.323, Z    +0.000, E1   -25.412, E3 -488251.249}
SPL {X  -159.990, Y  +451.400, Z    +0.000, E1   -25.397, E3 -488264.340}
SPL {X  -159.990, Y  +448.503, Z    +0.000, E1   -25.410, E3 -488277.257}
SPL {X  -159.990, Y  +445.882, Z    +0.000, E1   -25.385, E3 -488289.060}
SPL {X  -159.990, Y  +443.345, Z    +0.000, E1   -25.390, E3 -488300.442}
SPL {X  -159.990, Y  +441.077, Z    +0.000, E1   -25.369, E3 -488310.640}
SPL {X  -159.990, Y  +438.608, Z    +0.000, E1   -25.392, E3 -488321.637}
SPL {X  -159.990, Y  +434.852, Z    +0.000, E1   -25.415, E3 -488338.392}
SPL {X  -159.990, Y  +430.645, Z    +0.000, E1   -25.414, E3 -488357.211}
SPL {X  -159.990, Y  +426.865, Z    +0.000, E1   -25.398, E3 -488374.141}
SPL {X  -159.990, Y  +424.251, Z    +0.000, E1   -25.375, E3 -488385.878}
SPL {X  -159.990, Y  +421.010, Z    +0.000, E1   -25.418, E3 -488400.293}
SPL {X  -159.990, Y  +417.514, Z    +0.000, E1   -25.386, E3 -488415.986}
SPL {X  -159.990, Y  +414.805, Z    +0.000, E1   -25.385, E3 -488428.106}
SPL {X  -159.990, Y  +411.959, Z    +0.000, E1   -25.386, E3 -488440.832}
SPL {X  -159.990, Y  +408.981, Z    +0.000, E1   -25.392, E3 -488454.136}
SPL {X  -159.990, Y  +406.574, Z    +0.000, E1   -25.375, E3 -488464.910}
SPL {X  -159.990, Y  +403.513, Z    +0.000, E1   -25.420, E3 -488478.509}
SPL {X  -159.990, Y  +399.257, Z    +0.000, E1   -25.420, E3 -488497.550}
SPL {X  -159.990, Y  +395.992, Z    +0.000, E1   -25.380, E3 -488512.240}
SPL {X  -159.990, Y  +393.569, Z    +0.000, E1   -25.379, E3 -488523.083}
SPL {X  -159.990, Y  +390.564, Z    +0.000, E1   -25.393, E3 -488536.527}
SPL {X  -159.990, Y  +387.503, Z    +0.000, E1   -25.378, E3 -488550.242}
SPL {X  -159.990, Y  +384.900, Z    +0.000, E1   -25.383, E3 -488561.851}
SPL {X  -159.990, Y  +382.110, Z    +0.000, E1   -25.393, E3 -488574.298}
SPL {X  -159.961, Y  +379.439, Z    +0.000, E1   -25.380, E3 -488586.277}
SPL {X  -159.894, Y  +376.959, Z    +0.000, E1   -25.370, E3 -488597.455}
SPL {X  -159.784, Y  +374.382, Z    +0.000, E1   -25.356, E3 -488609.095}
SPL {X  -159.621, Y  +371.640, Z    +0.000, E1   -25.335, E3 -488621.535}
SPL {X  -159.406, Y  +368.844, Z    +0.000, E1   -25.307, E3 -488634.248}
SPL {X  -159.144, Y  +366.072, Z    +0.000, E1   -25.281, E3 -488646.856}
SPL {X  -158.822, Y  +363.200, Z    +0.000, E1   -25.236, E3 -488660.028}
SPL {X  -158.491, Y  +360.654, Z    +0.000, E1   -25.188, E3 -488671.769}
SPL {X  -158.127, Y  +358.155, Z    +0.000, E1   -25.126, E3 -488683.388}
SPL {X  -158.095, Y  +357.947, Z    +0.000, E1   -21.741, E3 -488714.960}
ENDSPLINE

SPLINE
SPL {X  -158.454, Y  +360.384, Z    +0.000, E1   -19.366, E3 -488727.111}
SPL {X  -159.737, Y  +373.507, Z    +0.000, E1   -10.311, E3 -488749.147}
SPL {X  -159.990, Y  +382.574, Z    +0.000, E1    -4.463, E3 -488755.835}
SPL {X  -159.990, Y  +389.909, Z    +0.000, E1    +0.662, E3 -488759.849}
SPL {X  -159.990, Y  +396.289, Z    +0.000, E1    +5.500, E3 -488763.629}
SPL {X  -159.990, Y  +407.941, Z    +0.000, E1   +14.126, E3 -488774.966}
SPL {X  -159.990, Y  +418.671, Z    +0.000, E1   +19.855, E3 -488794.382}
SPL {X  -159.990, Y  +429.878, Z    +0.000, E1   +23.330, E3 -488824.437}
SPL {X  -159.990, Y  +432.766, Z    +0.000, E1   +23.321, E3 -488838.660}
SPL {X  -159.990, Y  +434.794, Z    +0.000, E1   +23.304, E3 -488848.691}
SPL {X  -159.990, Y  +437.007, Z    +0.000, E1   +23.323, E3 -488859.544}
SPL {X  -159.990, Y  +439.778, Z    +0.000, E1   +23.323, E3 -488873.176}
SPL {X  -159.990, Y  +442.010, Z    +0.000, E1   +23.308, E3 -488884.197}
SPL {X  -159.990, Y  +443.729, Z    +0.000, E1   +23.310, E3 -488892.653}
SPL {X  -159.990, Y  +446.037, Z    +0.000, E1   +23.324, E3 -488903.990}
SPL {X  -159.990, Y  +449.434, Z    +0.000, E1   +23.356, E3 -488920.612}
SPL {X  -159.990, Y  +453.256, Z    +0.000, E1   +23.349, E3 -488939.447}
SPL {X  -159.990, Y  +455.953, Z    +0.000, E1   +23.320, E3 -488952.761}
SPL {X  -159.990, Y  +458.265, Z    +0.000, E1   +23.328, E3 -488964.115}
SPL {X  -159.990, Y  +460.492, Z    +0.000, E1   +23.317, E3 -488975.114}
SPL {X  -159.990, Y  +462.929, Z    +0.000, E1   +23.331, E3 -488987.070}
SPL {X  -159.990, Y  +466.197, Z    +0.000, E1   +23.351, E3 -489003.107}
SPL {X  -159.990, Y  +468.951, Z    +0.000, E1   +23.319, E3 -489016.725}
SPL {X  -159.990, Y  +470.991, Z    +0.000, E1   +23.322, E3 -489026.755}
SPL {X  -159.990, Y  +474.027, Z    +0.000, E1   +23.352, E3 -489041.658}
SPL {X  -159.990, Y  +477.600, Z    +0.000, E1   +23.351, E3 -489059.262}
SPL {X  -159.990, Y  +481.169, Z    +0.000, E1   +23.337, E3 -489076.859}
SPL {X  -159.990, Y  +483.782, Z    +0.000, E1   +23.316, E3 -489089.764}
SPL {X  -159.990, Y  +486.109, Z    +0.000, E1   +23.322, E3 -489101.216}
SPL {X  -159.990, Y  +489.247, Z    +0.000, E1   +23.348, E3 -489116.603}
SPL {X  -159.990, Y  +493.031, Z    +0.000, E1   +23.350, E3 -489135.228}
SPL {X  -159.990, Y  +496.869, Z    +0.000, E1   +23.349, E3 -489154.118}
SPL {X  -159.990, Y  +499.995, Z    +0.000, E1   +23.324, E3 -489169.551}
SPL {X  -159.990, Y  +502.456, Z    +0.000, E1   +23.324, E3 -489181.666}
SPL {X  -159.990, Y  +505.646, Z    +0.000, E1   +23.350, E3 -489197.321}
SPL {X  -159.990, Y  +508.862, Z    +0.000, E1   +23.328, E3 -489213.185}
SPL {X  -159.990, Y  +510.971, Z    +0.000, E1   +23.308, E3 -489223.613}
SPL {X  -159.990, Y  +513.289, Z    +0.000, E1   +23.332, E3 -489234.980}
SPL {X  -159.990, Y  +516.860, Z    +0.000, E1   +23.355, E3 -489252.497}
SPL {X  -159.990, Y  +520.719, Z    +0.000, E1   +23.363, E3 -489271.407}
SPL {X  -159.990, Y  +523.968, Z    +0.000, E1   +23.332, E3 -489287.492}
SPL {X  -159.990, Y  +526.466, Z    +0.000, E1   +23.320, E3 -489299.835}
SPL {X  -159.990, Y  +528.815, Z    +0.000, E1   +23.322, E3 -489311.395}
SPL {X  -159.990, Y  +531.246, Z    +0.000, E1   +23.325, E3 -489323.334}
SPL {X  -159.990, Y  +533.354, Z    +0.000, E1   +23.318, E3 -489333.719}
SPL {X  -159.990, Y  +534.931, Z    +0.000, E1   +23.312, E3 -489341.513}
SPL {X  -159.990, Y  +537.024, Z    +0.000, E1   +23.321, E3 -489351.812}
SPL {X  -159.990, Y  +539.129, Z    +0.000, E1   +23.310, E3 -489362.195}
SPL {X  -159.990, Y  +541.183, Z    +0.000, E1   +23.319, E3 -489372.292}
SPL {X  -159.990, Y  +544.314, Z    +0.000, E1   +23.352, E3 -489387.620}
SPL {X  -159.990, Y  +548.126, Z    +0.000, E1   +23.354, E3 -489406.375}
SPL {X  -159.990, Y  +551.344, Z    +0.000, E1   +23.327, E3 -489422.267}
SPL {X  -159.990, Y  +553.642, Z    +0.000, E1   +23.319, E3 -489433.586}
SPL {X  -159.990, Y  +556.481, Z    +0.000, E1   +23.354, E3 -489447.493}
SPL {X  -159.990, Y  +559.475, Z    +0.000, E1   +23.321, E3 -489462.298}
SPL {X  -159.990, Y  +561.830, Z    +0.000, E1   +23.325, E3 -489473.883}
SPL {X  -159.990, Y  +564.273, Z    +0.000, E1   +23.325, E3 -489485.907}
SPL {X  -159.990, Y  +566.342, Z    +0.000, E1   +23.314, E3 -489496.112}
SPL {X  -159.990, Y  +568.849, Z    +0.000, E1   +23.338, E3 -489508.407}
SPL {X  -159.990, Y  +572.204, Z    +0.000, E1   +23.344, E3 -489524.902}
SPL {X  -159.990, Y  +575.097, Z    +0.000, E1   +23.325, E3 -489539.179}
SPL {X  -159.990, Y  +577.540, Z    +0.000, E1   +23.325, E3 -489551.208}
SPL {X  -159.990, Y  +580.312, Z    +0.000, E1   +23.340, E3 -489564.789}
SPL {X  -159.990, Y  +583.018, Z    +0.000, E1   +23.331, E3 -489578.094}
SPL {X  -159.990, Y  +585.165, Z    +0.000, E1   +23.322, E3 -489588.710}
SPL {X  -159.990, Y  +587.388, Z    +0.000, E1   +23.328, E3 -489599.622}
SPL {X  -159.990, Y  +589.763, Z    +0.000, E1   +23.328, E3 -489611.309}
SPL {X  -159.990, Y  +592.397, Z    +0.000, E1   +23.344, E3 -489624.190}
SPL {X  -159.990, Y  +595.589, Z    +0.000, E1   +23.356, E3 -489639.863}
SPL {X  -159.990, Y  +598.571, Z    +0.000, E1   +23.347, E3 -489654.506}
SPL {X  -159.990, Y  +600.935, Z    +0.000, E1   +23.343, E3 -489666.099}
SPL {X  -159.990, Y  +603.047, Z    +0.000, E1   +23.344, E3 -489676.485}
SPL {X  -159.990, Y  +605.187, Z    +0.000, E1   +23.344, E3 -489687.007}
SPL {X  -159.990, Y  +607.319, Z    +0.000, E1   +23.353, E3 -489697.469}
SPL {X  -159.990, Y  +610.569, Z    +0.000, E1   +23.372, E3 -489713.434}
SPL {X  -159.990, Y  +613.591, Z    +0.000, E1   +23.342, E3 -489728.363}
SPL {X  -159.990, Y  +615.604, Z    +0.000, E1   +23.330, E3 -489738.301}
SPL {X  -159.990, Y  +618.445, Z    +0.000, E1   +23.368, E3 -489752.214}
SPL {X  -159.990, Y  +621.517, Z    +0.000, E1   +23.337, E3 -489767.378}
SPL {X  -159.990, Y  +623.764, Z    +0.000, E1   +23.335, E3 -489778.429}
SPL {X  -159.990, Y  +626.608, Z    +0.000, E1   +23.361, E3 -489792.354}
SPL {X  -159.990, Y  +630.271, Z    +0.000, E1   +23.375, E3 -489810.315}
SPL {X  -159.990, Y  +633.318, Z    +0.000, E1   +23.339, E3 -489825.392}
SPL {X  -159.990, Y  +635.650, Z    +0.000, E1   +23.339, E3 -489836.863}
SPL {X  -159.990, Y  +637.839, Z    +0.000, E1   +23.335, E3 -489847.674}
SPL {X  -159.990, Y  +640.072, Z    +0.000, E1   +23.325, E3 -489858.706}
SPL {X  -159.990, Y  +643.026, Z    +0.000, E1   +23.354, E3 -489873.246}
SPL {X  -159.990, Y  +646.970, Z    +0.000, E1   +23.346, E3 -489892.709}
SPL {X  -159.990, Y  +650.790, Z    +0.000, E1   +23.346, E3 -489911.498}
SPL {X  -159.990, Y  +654.543, Z    +0.000, E1   +23.348, E3 -489929.950}
SPL {X  -159.990, Y  +658.319, Z    +0.000, E1   +23.349, E3 -489948.540}
SPL {X  -159.990, Y  +661.392, Z    +0.000, E1   +23.318, E3 -489963.743}
SPL {X  -159.990, Y  +663.662, Z    +0.000, E1   +23.322, E3 -489974.867}
SPL {X  -159.990, Y  +665.964, Z    +0.000, E1   +23.328, E3 -489986.158}
SPL {X  -159.990, Y  +667.870, Z    +0.000, E1   +23.320, E3 -489995.565}
SPL {X  -159.990, Y  +669.861, Z    +0.000, E1   +23.321, E3 -490005.366}
SPL {X  -159.990, Y  +671.893, Z    +0.000, E1   +23.319, E3 -490015.374}
SPL {X  -159.974, Y  +673.789, Z    +0.000, E1   +23.323, E3 -490024.689}
SPL {X  -159.924, Y  +676.110, Z    +0.000, E1   +23.320, E3 -490036.174}
SPL {X  -159.801, Y  +679.265, Z    +0.000, E1   +23.327, E3 -490051.793}
SPL {X  -159.626, Y  +682.287, Z    +0.000, E1   +23.280, E3 -490066.891}
SPL {X  -159.462, Y  +684.486, Z    +0.000, E1   +23.258, E3 -490077.891}
SPL {X  -159.246, Y  +686.911, Z    +0.000, E1   +23.230, E3 -490090.052}
SPL {X  -159.019, Y  +689.098, Z    +0.000, E1   +23.200, E3 -490101.054}
SPL {X  -158.660, Y  +692.086, Z    +0.000, E1   +23.176, E3 -490116.098}
ENDSPLINE

SPLINE
SPL {X  -159.063, Y  +688.696, Z    +0.000, E1   +17.094, E3 -490158.379}
SPL {X  -159.967, Y  +674.206, Z    +0.000, E1    +6.731, E3 -490181.192}
SPL {X  -159.990, Y  +665.270, Z    +0.000, E1    +0.699, E3 -490187.362}
SPL {X  -159.990, Y  +658.009, Z    +0.000, E1    -4.774, E3 -490191.939}
SPL {X  -159.990, Y  +651.567, Z    +0.000, E1    -9.674, E3 -490197.342}
SPL {X  -159.990, Y  +637.762, Z    +0.000, E1   -18.345, E3 -490214.700}
SPL {X  -159.990, Y  +626.382, Z    +0.000, E1   -22.040, E3 -490246.749}
SPL {X  -159.990, Y  +623.760, Z    +0.000, E1   -22.031, E3 -490260.527}
SPL {X  -159.990, Y  +621.334, Z    +0.000, E1   -22.029, E3 -490273.254}
SPL {X  -159.990, Y  +618.387, Z    +0.000, E1   -22.057, E3 -490288.643}
SPL {X  -159.990, Y  +614.928, Z    +0.000, E1   -22.055, E3 -490306.796}
SPL {X  -159.990, Y  +611.459, Z    +0.000, E1   -22.053, E3 -490324.999}
SPL {X  -159.990, Y  +608.810, Z    +0.000, E1   -22.023, E3 -490338.967}
SPL {X  -159.990, Y  +606.481, Z    +0.000, E1   -22.033, E3 -490351.142}
SPL {X  -159.990, Y  +603.419, Z    +0.000, E1   -22.064, E3 -490367.082}
SPL {X  -159.990, Y  +600.642, Z    +0.000, E1   -22.032, E3 -490381.712}
SPL {X  -159.990, Y  +598.568, Z    +0.000, E1   -22.046, E3 -490392.504}
SPL {X  -159.990, Y  +596.440, Z    +0.000, E1   -22.036, E3 -490403.686}
SPL {X  -159.990, Y  +593.768, Z    +0.000, E1   -22.071, E3 -490417.619}
SPL {X  -159.990, Y  +590.068, Z    +0.000, E1   -22.076, E3 -490436.987}
SPL {X  -159.990, Y  +587.130, Z    +0.000, E1   -22.046, E3 -490452.424}
SPL {X  -159.990, Y  +585.120, Z    +0.000, E1   -22.045, E3 -490462.926}
SPL {X  -159.990, Y  +583.118, Z    +0.000, E1   -22.052, E3 -490473.412}
SPL {X  -159.990, Y  +580.862, Z    +0.000, E1   -22.049, E3 -490485.250}
SPL {X  -159.990, Y  +578.386, Z    +0.000, E1   -22.057, E3 -490498.205}
SPL {X  -159.990, Y  +576.252, Z    +0.000, E1   -22.038, E3 -490509.428}
SPL {X  -159.990, Y  +574.280, Z    +0.000, E1   -22.051, E3 -490519.722}
SPL {X  -159.990, Y  +571.711, Z    +0.000, E1   -22.058, E3 -490533.196}
SPL {X  -159.990, Y  +569.285, Z    +0.000, E1   -22.044, E3 -490545.921}
SPL {X  -159.990, Y  +567.211, Z    +0.000, E1   -22.046, E3 -490556.783}
SPL {X  -159.990, Y  +565.039, Z    +0.000, E1   -22.047, E3 -490568.160}
SPL {X  -159.990, Y  +562.755, Z    +0.000, E1   -22.047, E3 -490580.145}
SPL {X  -159.990, Y  +559.661, Z    +0.000, E1   -22.078, E3 -490596.277}
SPL {X  -159.990, Y  +555.965, Z    +0.000, E1   -22.085, E3 -490615.586}
SPL {X  -159.990, Y  +553.115, Z    +0.000, E1   -22.054, E3 -490630.571}
SPL {X  -159.990, Y  +550.886, Z    +0.000, E1   -22.056, E3 -490642.253}
SPL {X  -159.990, Y  +548.814, Z    +0.000, E1   -22.049, E3 -490653.099}
SPL {X  -159.990, Y  +546.122, Z    +0.000, E1   -22.088, E3 -490667.112}
SPL {X  -159.990, Y  +542.390, Z    +0.000, E1   -22.086, E3 -490686.694}
SPL {X  -159.990, Y  +539.341, Z    +0.000, E1   -22.056, E3 -490702.715}
SPL {X  -159.990, Y  +536.301, Z    +0.000, E1   -22.084, E3 -490718.570}
SPL {X  -159.990, Y  +533.389, Z    +0.000, E1   -22.057, E3 -490733.878}
SPL {X  -159.990, Y  +531.347, Z    +0.000, E1   -22.052, E3 -490744.578}
SPL {X  -159.990, Y  +528.972, Z    +0.000, E1   -22.072, E3 -490756.951}
SPL {X  -159.990, Y  +526.034, Z    +0.000, E1   -22.073, E3 -490772.330}
SPL {X  -159.990, Y  +523.717, Z    +0.000, E1   -22.050, E3 -490784.535}
SPL {X  -159.990, Y  +521.599, Z    +0.000, E1   -22.060, E3 -490795.603}
SPL {X  -159.990, Y  +519.209, Z    +0.000, E1   -22.063, E3 -490808.078}
SPL {X  -159.990, Y  +517.330, Z    +0.000, E1   -22.053, E3 -490817.934}
SPL {X  -159.990, Y  +514.729, Z    +0.000, E1   -22.089, E3 -490831.492}
SPL {X  -159.990, Y  +511.670, Z    +0.000, E1   -22.064, E3 -490847.579}
SPL {X  -159.990, Y  +506.947, Z    +0.000, E1   -23.726, E3 -490857.607}
SPL {X  -159.990, Y  +496.921, Z    +0.000, E1   -28.340, E3 -490866.356}
SPL {X  -159.990, Y  +495.822, Z    +0.000, E1   -27.449, E3 -490877.104}
SPL {X  -159.990, Y  +494.952, Z    +0.000, E1   -26.628, E3 -490886.687}
SPL {X  -159.990, Y  +493.896, Z    +0.000, E1   -25.736, E3 -490898.017}
SPL {X  -159.990, Y  +491.647, Z    +0.000, E1   -25.401, E3 -490910.552}
SPL {X  -159.990, Y  +488.807, Z    +0.000, E1   -25.397, E3 -490923.251}
SPL {X  -159.990, Y  +486.070, Z    +0.000, E1   -25.399, E3 -490935.482}
SPL {X  -159.990, Y  +482.821, Z    +0.000, E1   -25.411, E3 -490949.983}
SPL {X  -159.990, Y  +480.183, Z    +0.000, E1   -25.384, E3 -490961.824}
SPL {X  -159.990, Y  +477.508, Z    +0.000, E1   -25.410, E3 -490973.732}
SPL {X  -159.990, Y  +473.634, Z    +0.000, E1   -25.426, E3 -490991.021}
SPL {X  -159.990, Y  +470.047, Z    +0.000, E1   -25.402, E3 -491007.102}
SPL {X  -159.990, Y  +466.213, Z    +0.000, E1   -25.433, E3 -491024.182}
SPL {X  -159.990, Y  +462.520, Z    +0.000, E1   -25.400, E3 -491040.751}
SPL {X  -159.990, Y  +460.081, Z    +0.000, E1   -25.390, E3 -491051.652}
SPL {X  -159.990, Y  +457.497, Z    +0.000, E1   -25.403, E3 -491063.177}
SPL {X  -159.990, Y  +454.323, Z    +0.000, E1   -25.412, E3 -491077.336}
SPL {X  -159.990, Y  +451.400, Z    +0.000, E1   -25.397, E3 -491090.427}
SPL {X  -159.990, Y  +448.503, Z    +0.000, E1   -25.410, E3 -491103.344}
SPL {X  -159.990, Y  +445.108, Z    +0.000, E1   -25.407, E3 -491118.582}
SPL {X  -159.990, Y  +441.797, Z    +0.000, E1   -25.390, E3 -491133.461}
SPL {X  -159.990, Y  +439.442, Z    +0.000, E1   -25.369, E3 -491144.038}
SPL {X  -159.990, Y  +436.316, Z    +0.000, E1   -25.420, E3 -491157.920}
SPL {X  -159.990, Y  +432.613, Z    +0.000, E1   -25.390, E3 -491174.545}
SPL {X  -159.990, Y  +429.079, Z    +0.000, E1   -25.407, E3 -491190.316}
SPL {X  -159.990, Y  +426.149, Z    +0.000, E1   -25.374, E3 -491203.478}
SPL {X  -159.990, Y  +423.417, Z    +0.000, E1   -25.400, E3 -491215.644}
SPL {X  -159.990, Y  +420.283, Z    +0.000, E1   -25.386, E3 -491229.688}
SPL {X  -159.990, Y  +417.514, Z    +0.000, E1   -25.386, E3 -491242.073}
SPL {X  -159.990, Y  +414.805, Z    +0.000, E1   -25.385, E3 -491254.193}
SPL {X  -159.990, Y  +411.282, Z    +0.000, E1   -25.413, E3 -491269.893}
SPL {X  -159.990, Y  +408.351, Z    +0.000, E1   -25.372, E3 -491283.080}
SPL {X  -159.990, Y  +405.773, Z    +0.000, E1   -25.398, E3 -491294.533}
SPL {X  -159.990, Y  +402.805, Z    +0.000, E1   -25.389, E3 -491307.819}
SPL {X  -159.990, Y  +400.083, Z    +0.000, E1   -25.388, E3 -491319.996}
SPL {X  -159.990, Y  +396.740, Z    +0.000, E1   -25.410, E3 -491334.920}
SPL {X  -159.990, Y  +392.622, Z    +0.000, E1   -25.413, E3 -491353.348}
SPL {X  -159.990, Y  +388.328, Z    +0.000, E1   -25.413, E3 -491372.576}
SPL {X  -159.990, Y  +384.900, Z    +0.000, E1   -25.383, E3 -491387.938}
SPL {X  -159.990, Y  +382.110, Z    +0.000, E1   -25.393, E3 -491400.385}
SPL {X  -159.961, Y  +379.439, Z    +0.000, E1   -25.380, E3 -491412.364}
SPL {X  -159.894, Y  +376.959, Z    +0.000, E1   -25.370, E3 -491423.542}
SPL {X  -159.784, Y  +374.382, Z    +0.000, E1   -25.356, E3 -491435.182}
SPL {X  -159.621, Y  +371.640, Z    +0.000, E1   -25.335, E3 -491447.622}
SPL {X  -159.406, Y  +368.844, Z    +0.000, E1   -25.307, E3 -491460.335}
SPL {X  -159.144, Y  +366.072, Z    +0.000, E1   -25.281, E3 -491472.943}
SPL {X  -158.822, Y  +363.200, Z    +0.000, E1   -25.236, E3 -491486.115}
SPL {X  -158.491, Y  +360.654, Z    +0.000, E1   -25.188, E3 -491497.856}
SPL {X  -158.127, Y  +358.155, Z    +0.000, E1   -25.126, E3 -491509.475}
SPL {X  -158.095, Y  +357.947, Z    +0.000, E1   -21.741, E3 -491541.047}
ENDSPLINE

SPLINE
SPL {X  -158.454, Y  +360.384, Z    +0.000, E1   -19.366, E3 -491553.198}
SPL {X  -159.737, Y  +373.507, Z    +0.000, E1   -10.311, E3 -491575.234}
SPL {X  -159.990, Y  +382.574, Z    +0.000, E1    -4.463, E3 -491581.921}
SPL {X  -159.990, Y  +389.909, Z    +0.000, E1    +0.662, E3 -491585.936}
SPL {X  -159.990, Y  +396.289, Z    +0.000, E1    +5.500, E3 -491589.716}
SPL {X  -159.990, Y  +407.941, Z    +0.000, E1   +14.126, E3 -491601.053}
SPL {X  -159.990, Y  +418.671, Z    +0.000, E1   +19.855, E3 -491620.469}
SPL {X  -159.990, Y  +429.878, Z    +0.000, E1   +23.330, E3 -491650.524}
SPL {X  -159.990, Y  +432.766, Z    +0.000, E1   +23.321, E3 -491664.747}
SPL {X  -159.990, Y  +434.794, Z    +0.000, E1   +23.304, E3 -491674.778}
SPL {X  -159.990, Y  +437.007, Z    +0.000, E1   +23.323, E3 -491685.631}
SPL {X  -159.990, Y  +439.778, Z    +0.000, E1   +23.323, E3 -491699.263}
SPL {X  -159.990, Y  +442.945, Z    +0.000, E1   +23.339, E3 -491714.827}
SPL {X  -159.990, Y  +446.037, Z    +0.000, E1   +23.324, E3 -491730.077}
SPL {X  -159.990, Y  +448.797, Z    +0.000, E1   +23.331, E3 -491743.608}
SPL {X  -159.990, Y  +451.747, Z    +0.000, E1   +23.333, E3 -491758.155}
SPL {X  -159.990, Y  +455.185, Z    +0.000, E1   +23.350, E3 -491775.015}
SPL {X  -159.990, Y  +458.265, Z    +0.000, E1   +23.328, E3 -491790.202}
SPL {X  -159.990, Y  +461.258, Z    +0.000, E1   +23.344, E3 -491804.918}
SPL {X  -159.990, Y  +464.382, Z    +0.000, E1   +23.332, E3 -491820.299}
SPL {X  -159.990, Y  +466.881, Z    +0.000, E1   +23.322, E3 -491832.620}
SPL {X  -159.990, Y  +468.951, Z    +0.000, E1   +23.319, E3 -491842.812}
SPL {X  -159.990, Y  +470.991, Z    +0.000, E1   +23.322, E3 -491852.842}
SPL {X  -159.990, Y  +474.027, Z    +0.000, E1   +23.352, E3 -491867.745}
SPL {X  -159.990, Y  +476.830, Z    +0.000, E1   +23.323, E3 -491881.613}
SPL {X  -159.990, Y  +479.553, Z    +0.000, E1   +23.328, E3 -491895.015}
SPL {X  -159.990, Y  +482.950, Z    +0.000, E1   +23.350, E3 -491911.687}
SPL {X  -159.990, Y  +486.109, Z    +0.000, E1   +23.322, E3 -491927.303}
SPL {X  -159.990, Y  +488.481, Z    +0.000, E1   +23.319, E3 -491938.983}
SPL {X  -159.990, Y  +491.454, Z    +0.000, E1   +23.343, E3 -491953.563}
SPL {X  -159.990, Y  +493.986, Z    +0.000, E1   +23.312, E3 -491966.092}
SPL {X  -159.990, Y  +496.869, Z    +0.000, E1   +23.349, E3 -491980.205}
SPL {X  -159.990, Y  +499.995, Z    +0.000, E1   +23.324, E3 -491995.638}
SPL {X  -159.990, Y  +502.456, Z    +0.000, E1   +23.324, E3 -492007.753}
SPL {X  -159.990, Y  +505.646, Z    +0.000, E1   +23.350, E3 -492023.408}
SPL {X  -159.990, Y  +508.862, Z    +0.000, E1   +23.328, E3 -492039.272}
SPL {X  -159.990, Y  +510.971, Z    +0.000, E1   +23.308, E3 -492049.700}
SPL {X  -159.990, Y  +512.484, Z    +0.000, E1   +23.309, E3 -492057.149}
SPL {X  -159.990, Y  +514.757, Z    +0.000, E1   +23.329, E3 -492068.302}
SPL {X  -159.990, Y  +517.536, Z    +0.000, E1   +23.326, E3 -492081.968}
SPL {X  -159.990, Y  +519.961, Z    +0.000, E1   +23.334, E3 -492093.821}
SPL {X  -159.990, Y  +521.849, Z    +0.000, E1   +23.320, E3 -492103.143}
SPL {X  -159.990, Y  +523.968, Z    +0.000, E1   +23.332, E3 -492113.579}
SPL {X  -159.990, Y  +526.466, Z    +0.000, E1   +23.320, E3 -492125.922}
SPL {X  -159.990, Y  +528.815, Z    +0.000, E1   +23.322, E3 -492137.482}
SPL {X  -159.990, Y  +531.246, Z    +0.000, E1   +23.325, E3 -492149.421}
SPL {X  -159.990, Y  +534.143, Z    +0.000, E1   +23.341, E3 -492163.656}
SPL {X  -159.990, Y  +537.024, Z    +0.000, E1   +23.321, E3 -492177.899}
SPL {X  -159.990, Y  +539.129, Z    +0.000, E1   +23.310, E3 -492188.282}
SPL {X  -159.990, Y  +541.882, Z    +0.000, E1   +23.346, E3 -492201.763}
SPL {X  -159.990, Y  +544.941, Z    +0.000, E1   +23.325, E3 -492216.845}
SPL {X  -159.990, Y  +547.390, Z    +0.000, E1   +23.325, E3 -492228.899}
SPL {X  -159.990, Y  +550.708, Z    +0.000, E1   +23.357, E3 -492245.166}
SPL {X  -159.990, Y  +553.642, Z    +0.000, E1   +23.319, E3 -492259.673}
SPL {X  -159.990, Y  +555.637, Z    +0.000, E1   +23.323, E3 -492269.487}
SPL {X  -159.990, Y  +558.758, Z    +0.000, E1   +23.351, E3 -492284.797}
SPL {X  -159.990, Y  +561.830, Z    +0.000, E1   +23.325, E3 -492299.970}
SPL {X  -159.990, Y  +564.273, Z    +0.000, E1   +23.325, E3 -492311.994}
SPL {X  -159.990, Y  +567.351, Z    +0.000, E1   +23.348, E3 -492327.090}
SPL {X  -159.990, Y  +570.560, Z    +0.000, E1   +23.333, E3 -492342.920}
SPL {X  -159.990, Y  +572.975, Z    +0.000, E1   +23.316, E3 -492354.839}
SPL {X  -159.990, Y  +575.097, Z    +0.000, E1   +23.325, E3 -492365.266}
SPL {X  -159.990, Y  +577.540, Z    +0.000, E1   +23.325, E3 -492377.295}
SPL {X  -159.990, Y  +580.312, Z    +0.000, E1   +23.340, E3 -492390.876}
SPL {X  -159.990, Y  +583.018, Z    +0.000, E1   +23.331, E3 -492404.181}
SPL {X  -159.990, Y  +585.165, Z    +0.000, E1   +23.322, E3 -492414.797}
SPL {X  -159.990, Y  +587.388, Z    +0.000, E1   +23.328, E3 -492425.709}
SPL {X  -159.990, Y  +589.763, Z    +0.000, E1   +23.328, E3 -492437.396}
SPL {X  -159.990, Y  +592.397, Z    +0.000, E1   +23.344, E3 -492450.277}
SPL {X  -159.990, Y  +594.928, Z    +0.000, E1   +23.334, E3 -492462.739}
SPL {X  -159.990, Y  +597.981, Z    +0.000, E1   +23.373, E3 -492477.654}
SPL {X  -159.990, Y  +600.935, Z    +0.000, E1   +23.343, E3 -492492.186}
SPL {X  -159.990, Y  +603.047, Z    +0.000, E1   +23.344, E3 -492502.572}
SPL {X  -159.990, Y  +605.187, Z    +0.000, E1   +23.344, E3 -492513.094}
SPL {X  -159.990, Y  +607.319, Z    +0.000, E1   +23.353, E3 -492523.556}
SPL {X  -159.990, Y  +610.569, Z    +0.000, E1   +23.372, E3 -492539.521}
SPL {X  -159.990, Y  +613.591, Z    +0.000, E1   +23.342, E3 -492554.450}
SPL {X  -159.990, Y  +615.604, Z    +0.000, E1   +23.330, E3 -492564.388}
SPL {X  -159.990, Y  +618.445, Z    +0.000, E1   +23.368, E3 -492578.301}
SPL {X  -159.990, Y  +621.517, Z    +0.000, E1   +23.337, E3 -492593.465}
SPL {X  -159.990, Y  +623.764, Z    +0.000, E1   +23.335, E3 -492604.516}
SPL {X  -159.990, Y  +626.608, Z    +0.000, E1   +23.361, E3 -492618.441}
SPL {X  -159.990, Y  +630.271, Z    +0.000, E1   +23.375, E3 -492636.402}
SPL {X  -159.990, Y  +633.318, Z    +0.000, E1   +23.339, E3 -492651.479}
SPL {X  -159.990, Y  +635.650, Z    +0.000, E1   +23.339, E3 -492662.950}
SPL {X  -159.990, Y  +637.839, Z    +0.000, E1   +23.335, E3 -492673.760}
SPL {X  -159.990, Y  +640.072, Z    +0.000, E1   +23.325, E3 -492684.792}
SPL {X  -159.990, Y  +642.230, Z    +0.000, E1   +23.323, E3 -492695.474}
SPL {X  -159.990, Y  +645.287, Z    +0.000, E1   +23.340, E3 -492710.500}
SPL {X  -159.990, Y  +648.792, Z    +0.000, E1   +23.346, E3 -492727.759}
SPL {X  -159.990, Y  +652.623, Z    +0.000, E1   +23.348, E3 -492746.594}
SPL {X  -159.990, Y  +656.380, Z    +0.000, E1   +23.347, E3 -492765.088}
SPL {X  -159.990, Y  +659.180, Z    +0.000, E1   +23.314, E3 -492778.936}
SPL {X  -159.990, Y  +661.392, Z    +0.000, E1   +23.318, E3 -492789.830}
SPL {X  -159.990, Y  +663.662, Z    +0.000, E1   +23.322, E3 -492800.954}
SPL {X  -159.990, Y  +665.964, Z    +0.000, E1   +23.328, E3 -492812.245}
SPL {X  -159.990, Y  +668.989, Z    +0.000, E1   +23.359, E3 -492827.081}
SPL {X  -159.983, Y  +672.946, Z    +0.000, E1   +23.359, E3 -492846.562}
SPL {X  -159.924, Y  +676.110, Z    +0.000, E1   +23.320, E3 -492862.261}
SPL {X  -159.845, Y  +678.302, Z    +0.000, E1   +23.298, E3 -492873.163}
SPL {X  -159.760, Y  +680.081, Z    +0.000, E1   +23.288, E3 -492882.007}
SPL {X  -159.626, Y  +682.287, Z    +0.000, E1   +23.280, E3 -492892.978}
SPL {X  -159.462, Y  +684.486, Z    +0.000, E1   +23.258, E3 -492903.978}
SPL {X  -159.246, Y  +686.911, Z    +0.000, E1   +23.230, E3 -492916.139}
SPL {X  -159.019, Y  +689.098, Z    +0.000, E1   +23.200, E3 -492927.141}
SPL {X  -158.660, Y  +692.086, Z    +0.000, E1   +23.176, E3 -492942.185}
ENDSPLINE

SPLINE
SPL {X  -159.063, Y  +688.696, Z    +0.000, E1   +17.094, E3 -492984.466}
SPL {X  -159.967, Y  +674.206, Z    +0.000, E1    +6.731, E3 -493007.279}
SPL {X  -159.990, Y  +665.270, Z    +0.000, E1    +0.699, E3 -493013.449}
SPL {X  -159.990, Y  +658.009, Z    +0.000, E1    -4.774, E3 -493018.026}
SPL {X  -159.990, Y  +651.567, Z    +0.000, E1    -9.674, E3 -493023.429}
SPL {X  -159.990, Y  +638.711, Z    +0.000, E1   -17.883, E3 -493039.075}
SPL {X  -159.990, Y  +631.642, Z    +0.000, E1   -20.884, E3 -493054.634}
SPL {X  -159.990, Y  +626.048, Z    +0.000, E1   -22.026, E3 -493074.627}
SPL {X  -159.990, Y  +623.760, Z    +0.000, E1   -22.031, E3 -493086.614}
SPL {X  -159.990, Y  +621.334, Z    +0.000, E1   -22.029, E3 -493099.340}
SPL {X  -159.990, Y  +619.505, Z    +0.000, E1   -22.018, E3 -493108.956}
SPL {X  -159.990, Y  +617.621, Z    +0.000, E1   -22.025, E3 -493118.822}
SPL {X  -159.990, Y  +615.830, Z    +0.000, E1   -22.023, E3 -493128.222}
SPL {X  -159.990, Y  +613.034, Z    +0.000, E1   -22.053, E3 -493142.828}
SPL {X  -159.990, Y  +609.503, Z    +0.000, E1   -22.054, E3 -493161.355}
SPL {X  -159.990, Y  +605.804, Z    +0.000, E1   -22.064, E3 -493180.699}
SPL {X  -159.990, Y  +602.819, Z    +0.000, E1   -22.037, E3 -493196.370}
SPL {X  -159.990, Y  +600.642, Z    +0.000, E1   -22.032, E3 -493207.798}
SPL {X  -159.990, Y  +598.568, Z    +0.000, E1   -22.046, E3 -493218.591}
SPL {X  -159.990, Y  +595.493, Z    +0.000, E1   -22.070, E3 -493234.674}
SPL {X  -159.990, Y  +592.865, Z    +0.000, E1   -22.036, E3 -493248.503}
SPL {X  -159.990, Y  +590.803, Z    +0.000, E1   -22.046, E3 -493259.294}
SPL {X  -159.990, Y  +587.778, Z    +0.000, E1   -22.073, E3 -493275.069}
SPL {X  -159.990, Y  +585.120, Z    +0.000, E1   -22.045, E3 -493289.013}
SPL {X  -159.990, Y  +583.118, Z    +0.000, E1   -22.052, E3 -493299.499}
SPL {X  -159.990, Y  +580.131, Z    +0.000, E1   -22.078, E3 -493315.106}
SPL {X  -159.990, Y  +576.888, Z    +0.000, E1   -22.061, E3 -493332.136}
SPL {X  -159.990, Y  +574.280, Z    +0.000, E1   -22.051, E3 -493345.809}
SPL {X  -159.990, Y  +572.375, Z    +0.000, E1   -22.037, E3 -493355.848}
SPL {X  -159.990, Y  +569.881, Z    +0.000, E1   -22.067, E3 -493368.842}
SPL {X  -159.990, Y  +567.211, Z    +0.000, E1   -22.046, E3 -493382.869}
SPL {X  -159.990, Y  +565.039, Z    +0.000, E1   -22.047, E3 -493394.247}
SPL {X  -159.990, Y  +562.755, Z    +0.000, E1   -22.047, E3 -493406.232}
SPL {X  -159.990, Y  +560.652, Z    +0.000, E1   -22.038, E3 -493417.277}
SPL {X  -159.990, Y  +558.852, Z    +0.000, E1   -22.046, E3 -493426.649}
SPL {X  -159.990, Y  +556.672, Z    +0.000, E1   -22.055, E3 -493438.039}
SPL {X  -159.990, Y  +553.726, Z    +0.000, E1   -22.080, E3 -493453.401}
SPL {X  -159.990, Y  +550.886, Z    +0.000, E1   -22.056, E3 -493468.340}
SPL {X  -159.990, Y  +548.814, Z    +0.000, E1   -22.049, E3 -493479.186}
SPL {X  -159.990, Y  +546.122, Z    +0.000, E1   -22.088, E3 -493493.199}
SPL {X  -159.990, Y  +542.390, Z    +0.000, E1   -22.086, E3 -493512.781}
SPL {X  -159.990, Y  +539.341, Z    +0.000, E1   -22.056, E3 -493528.802}
SPL {X  -159.990, Y  +536.301, Z    +0.000, E1   -22.084, E3 -493544.657}
SPL {X  -159.990, Y  +533.389, Z    +0.000, E1   -22.057, E3 -493559.964}
SPL {X  -159.990, Y  +531.347, Z    +0.000, E1   -22.052, E3 -493570.665}
SPL {X  -159.990, Y  +529.626, Z    +0.000, E1   -22.051, E3 -493579.662}
SPL {X  -159.990, Y  +527.412, Z    +0.000, E1   -22.067, E3 -493591.215}
SPL {X  -159.990, Y  +524.425, Z    +0.000, E1   -22.078, E3 -493606.848}
SPL {X  -159.990, Y  +521.599, Z    +0.000, E1   -22.060, E3 -493621.690}
SPL {X  -159.990, Y  +519.209, Z    +0.000, E1   -22.063, E3 -493634.165}
SPL {X  -159.990, Y  +516.651, Z    +0.000, E1   -22.071, E3 -493647.544}
SPL {X  -159.990, Y  +514.122, Z    +0.000, E1   -22.061, E3 -493660.816}
SPL {X  -159.990, Y  +511.670, Z    +0.000, E1   -22.064, E3 -493673.666}
SPL {X  -159.990, Y  +506.947, Z    +0.000, E1   -23.726, E3 -493683.694}
SPL {X  -159.990, Y  +496.921, Z    +0.000, E1   -28.340, E3 -493692.443}
SPL {X  -159.990, Y  +495.822, Z    +0.000, E1   -27.449, E3 -493703.191}
SPL {X  -159.990, Y  +494.952, Z    +0.000, E1   -26.628, E3 -493712.774}
SPL {X  -159.990, Y  +493.896, Z    +0.000, E1   -25.736, E3 -493724.104}
ENDSPLINE

SLIN {X  -200.000, Y  +530.000, E1    +0.000}
HALT
END
